// TIA Portal V17 export
// export: Created 2022-07-20T06:59:48.3696304Z, ExportSetting WithDefaults, DisplayName Totally Integrated Automation Portal, DisplayVersion V17, DisplayName TIA Portal Openness, DisplayVersion V17, DisplayName TIA Portal Version Control Interface, DisplayVersion V17, DisplayName SINAMICS Startdrive Advanced, DisplayVersion V17, DisplayName SINAMICS Startdrive G130, G150, S120, S150, SINAMICS MV, S210, DisplayVersion V17, DisplayName SINAMICS Startdrive G110M, G120, G120C, G120D, G120P, G115D, DisplayVersion V17, DisplayName STEP 7 Professional, DisplayVersion V17, DisplayName STEP 7 Safety, DisplayVersion V17, DisplayName WinCC Advanced, DisplayVersion V17
FUNCTION "FC10206_AcknowledgeMachineAlarmStructure" : Void   // FC10206, LAD
{ S7_Optimized_Access := 'TRUE' }
VERSION : 0.1
// stored: AutoNumber false, IsIECCheckEnabled false, SetENOAutomatically false, UDAEnableTagReadback false
   VAR_INPUT
      Acknowledge : Bool;
   END_VAR
   VAR_OUTPUT
      AlarmStructure : "stStandardMgiMachineAlarms";
   END_VAR
BEGIN

REGION Network 1 (SCL)
   IF #Acknowledge THEN
       #AlarmStructure.ESTOP_Detected := FALSE;
       #AlarmStructure.STOP_Detected := FALSE;
       #AlarmStructure.HOLD_Detected := FALSE;
       #AlarmStructure.INFO_Detected := FALSE;
       #AlarmStructure.ESTOP_FirstAlarm := '';
       #AlarmStructure.STOP_FirstAlarm := '';
       #AlarmStructure.HOLD_FirstAlarm := '';
       #AlarmStructure.INFO_FirstAlarm := '';
   END_IF;
END_REGION
END_FUNCTION
